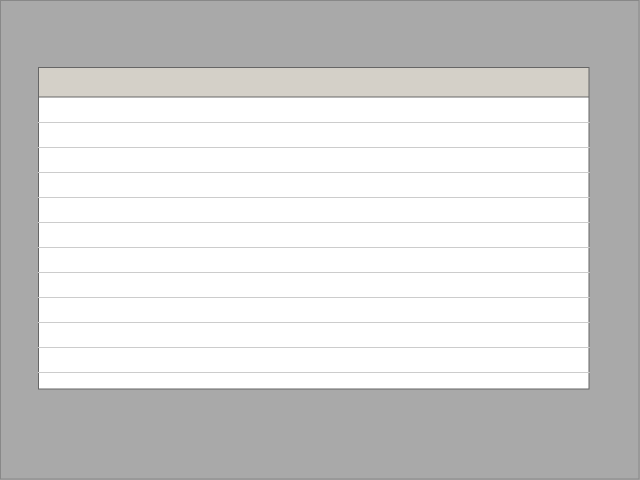
VISUALIZATION PH_ControllerInfo  // 640x480
VAR_IN_OUT
	strTargetType							: STRING(20);
	strHardwareModel						: STRING(10);
	strHardwareSerialNo						: STRING(12);
	strHardwareVersion						: STRING(4);
	strHardwareDate							: STRING(10);
	strHardwareCPU							: STRING(10);
	strImageDevice							: STRING(20);
	strImageVersion							: STRING(10);
	strImageLevel							: STRING(10);
	strImageOsName							: STRING(20);
	strImageOsVersion						: STRING(8);
	strTwinCATVersion						: STRING(4);
	strTwinCATRevision						: STRING(4);
	strTwinCATBuild							: STRING(8);
	strTwinCATLevel							: STRING(20);
	strAmsNetId								: STRING(23);
	arrDevIdent								: ARRAY [0..1, 1..16] OF STRING(23) ;
	wDeviceInfo								: WORD;
	iSelectedRow							: INT;
END_VAR
    Table (38,67 551x322), data array: arrDevIdent
        p338671338: MAIN.fbAutostartVisu.stDevIdent.strHardwareSerialNo
        p2170511999: MAIN.fbAutostartVisu.stDevIdent.strHardwareVersion
        p3723444502: MAIN.fbAutostartVisu.stDevIdent.strHardwareDate
        p1218418051: MAIN.fbAutostartVisu.stDevIdent.strHardwareCPU
        p746581629: MAIN.fbAutostartVisu.stDevIdent.strImageDevice
        p3104783080: MAIN.fbAutostartVisu.stDevIdent.strImageVersion
        p2501879983: MAIN.fbAutostartVisu.stDevIdent.strImageLevel
        p7306298: MAIN.fbAutostartVisu.stDevIdent.strImageOsName
        p1933151965: MAIN.fbAutostartVisu.stDevIdent.strImageOsVersion
        p3863566920: MAIN.fbAutostartVisu.stDevIdent.strTwinCATVersion
        p2192122294: MAIN.fbAutostartVisu.stDevIdent.strTwinCATRevision
        p400160035: MAIN.fbAutostartVisu.stDevIdent.strTwinCATBuild
        p1265227338: MAIN.fbAutostartVisu.stDevIdent.strTwinCATLevel
        p3726181087: MAIN.fbAutostartVisu.stDevIdent.strAmsNetId
        p3854506369: arrDevIdent[0,INDEX]
        p1892666644: arrDevIdent[1,INDEX]
        p1137915858: iSelectedRow
END_VISUALIZATION

(* stored: Version 1.1.0.1, ProductVersion 3.1.4024.3
   Visu PH_ControllerInfo: Id {515a96b4-d695-43f3-98fb-1aecd1365a78} *)
